DATA_BLOCK "ST10_PM"
VAR
  Num : Array[1..32] of "RCS_PMInterface_V1";
  Status : Array[1..50] of Int;
END_VAR
BEGIN
END_DATA_BLOCK
